Fanuc TP program (LS listing): UP112.LS

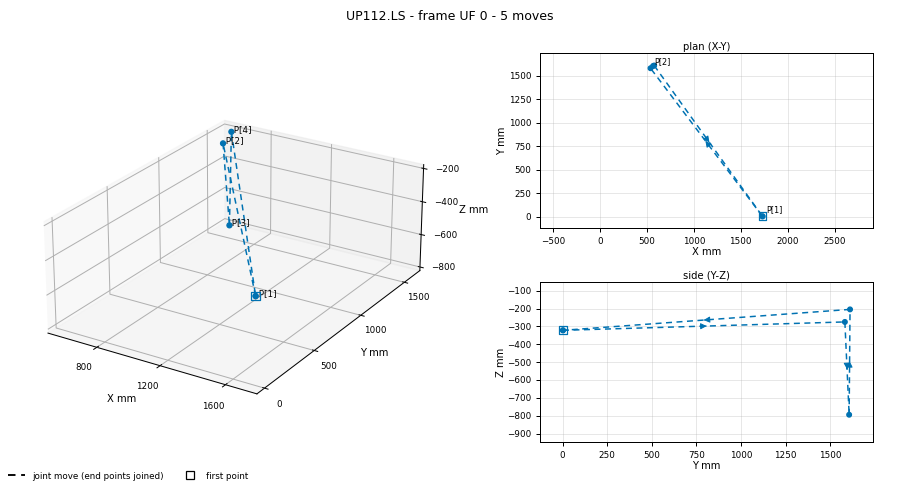
[picture p0: tool path of UP112.LS in frame UF 0, 5 of 5 moves have a stored position in this frame; points joined in program order, loops and branches not executed]
/PROG  UP112
/ATTR
OWNER		= AUROM;
COMMENT		= "Mantenimiento";
PROG_SIZE	= 2618;
CREATE		= DATE 03-15-00  TIME 13:37:40;
MODIFIED	= DATE 23-12-23  TIME 09:19:20;
FILE_NAME	= ;
VERSION		= 0;
LINE_COUNT	= 9;
MEMORY_SIZE	= 4830;
PROTECT		= READ_WRITE;
TCD:  STACK_SIZE	= 500,
      TASK_PRIORITY	= 50,
      TIME_SLICE	= 0,
      BUSY_LAMP_OFF	= 0,
      ABORT_REQUEST	= 0,
      PAUSE_REQUEST	= 0;
DEFAULT_GROUP	= 1,1,1,1,*;
CONTROL_CODE	= 00000000 00000000;
/MN
   1:  UTOOL_NUM=1 ;
   2:  UFRAME_NUM=0 ;
   3:  PAYLOAD[1] ;
   4:J P[1] 100% CNT0 ACC100 TB    .10sec,P-SPS    ;
      1:  TC_ONLINE (ON) ;
      2:  DO[23]=OFF ;
      3:  CALL MAKRO050    ;
      4:  !lib. de Herramientas ;
      5:  DO[80]=ON ;
      6:  !Lib. de Anticolisiones ;
      7:  DO[41]=ON ;
      8:  DO[42]=ON ;
      9:  DO[45]=ON ;
     10:  DO[46]=ON ;
     11:  !Apagar Posicion Base ;
     12:  DO[15]=OFF ;
     13:  WAIT (DI[23])    ;
     14:  DO[23]=ON ;
     15:  TC_ONLINE (M[30] AND M[95]) ;
       ------ ;
   5:J P[2] 100% CNT100 ACC100 TB   0.00sec,P-SPS    ;
      1:  TC_ONLINE (M[30] AND M[95]) ;
       ------ ;
   6:  !Posicion de Mantenimiento ;
   7:J P[3] 100% CNT0 ACC100 TB    .10sec,P-SPS    ;
      1:  TC_ONLINE (ON) ;
      2:  DO[23]=OFF ;
      3:  F[281]=(ON) ;
      4:  F[64]=(ON) ;
      5:  F[65]=(OFF) ;
      6:  F[66]=(OFF) ;
      7:  F[67]=(OFF) ;
      8:  CALL MAKRO089    ;
      9:  DO[17]=ON ;
     10:  GO[19]=(11) ;
     11:  WAIT (DI[17])    ;
     12:  IF (DI[132] AND !DI[133] AND !DI[134] AND !DI[135]),CALL MAKRO081 ;
     13:  LBL[1] ;
     14:  WAIT (!F[85] OR DI[26])    ;
     15:  IF (F[85]),CALL MAKRO081 ;
     16:  IF (F[85]),JMP LBL[1] ;
     17:  DO[17]=OFF ;
     18:  GO[19]=(0) ;
     19:  F[281]=(OFF) ;
     20:  WAIT (!DI[132] AND !DI[133] AND !DI[134] AND !DI[135])    ;
     21:  WAIT (DI[23])    ;
     22:  DO[23]=ON ;
     23:  TC_ONLINE (M[30] AND M[95]) ;
       ------ ;
   8:J P[4] 100% CNT100 ACC100 TB   0.00sec,P-SPS    ;
      1:  TC_ONLINE (M[30] AND M[95]) ;
       ------ ;
   9:J P[5] 100% CNT0 ACC100 TB    .10sec,P-SPS    ;
      1:  TC_ONLINE (ON) ;
      2:  DO[23]=OFF ;
      3:  WAIT (DI[23])    ;
      4:  DO[23]=ON ;
      5:  TC_ONLINE (M[30] AND M[95]) ;
       ------ ;
/POS
P[1]{
   GP1:
	UF : 0, UT : 1,		CONFIG : 'F U T, 0, 1, 0',
	X =  1731.500  mm,	Y =     2.242  mm,	Z =  -321.863  mm,
	W =  -176.060 deg,	P =    33.147 deg,	R =  -172.829 deg
   GP2:
	UF : 0, UT : 1,
	J1=   300.000  mm
   GP3:
	UF : 0, UT : 1,
	J1=     0.000  mm
   GP4:
	UF : 0, UT : 1,
	J1=     0.000  mm
};
P[2]{
   GP1:
	UF : 0, UT : 1,		CONFIG : 'F U T, 0, 0, 0',
	X =   537.687  mm,	Y =  1581.167  mm,	Z =  -274.929  mm,
	W =  -178.477 deg,	P =    16.515 deg,	R =  -100.139 deg
   GP2:
	UF : 0, UT : 1,
	J1=   298.200  mm
   GP3:
	UF : 0, UT : 1,
	J1=     0.000  mm
   GP4:
	UF : 0, UT : 1,
	J1=     0.000  mm
};
P[3]{
   GP1:
	UF : 0, UT : 1,		CONFIG : 'F U T, 0, 0, 0',
	X =   565.355  mm,	Y =  1605.108  mm,	Z =  -794.731  mm,
	W =  -178.346 deg,	P =    17.185 deg,	R =  -100.743 deg
   GP2:
	UF : 0, UT : 1,
	J1=   298.216  mm
   GP3:
	UF : 0, UT : 1,
	J1=     0.000  mm
   GP4:
	UF : 0, UT : 1,
	J1=     0.000  mm
};
P[4]{
   GP1:
	UF : 0, UT : 1,		CONFIG : 'F U T, 0, 0, 0',
	X =   576.832  mm,	Y =  1610.082  mm,	Z =  -204.716  mm,
	W =  -178.298 deg,	P =    17.394 deg,	R =  -101.042 deg
   GP2:
	UF : 0, UT : 1,
	J1=   298.224  mm
   GP3:
	UF : 0, UT : 1,
	J1=     0.000  mm
   GP4:
	UF : 0, UT : 1,
	J1=     0.000  mm
};
P[5]{
   GP1:
	UF : 0, UT : 1,		CONFIG : 'F U T, 0, 1, 0',
	X =  1731.500  mm,	Y =     2.242  mm,	Z =  -321.863  mm,
	W =  -176.060 deg,	P =    33.147 deg,	R =  -172.829 deg
   GP2:
	UF : 0, UT : 1,
	J1=   300.000  mm
   GP3:
	UF : 0, UT : 1,
	J1=     0.000  mm
   GP4:
	UF : 0, UT : 1,
	J1=     0.000  mm
};
/END
